FUNCTION_BLOCK HS_model
  (* Version 1.0, 2005-09-21, Goran Cengic, Chalmers *)
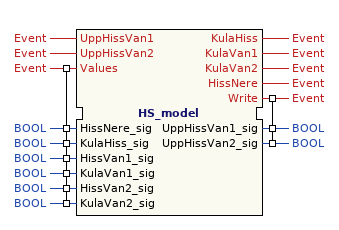
  EVENT_INPUT
    UppHissVan1;
    UppHissVan2;
    Values WITH KulaHiss_sig, HissVan1_sig, KulaVan1_sig, HissVan2_sig, KulaVan2_sig, HissNere_sig;
  END_EVENT
  EVENT_OUTPUT
    KulaHiss;
    KulaVan1;
    KulaVan2;
    HissNere;
    Write WITH UppHissVan1_sig, UppHissVan2_sig;
  END_EVENT
  VAR_INPUT
    HissNere_sig : BOOL;
    KulaHiss_sig : BOOL;
    HissVan1_sig : BOOL;
    KulaVan1_sig : BOOL;
    HissVan2_sig : BOOL;
    KulaVan2_sig : BOOL;
  END_VAR
  VAR_OUTPUT
    UppHissVan1_sig : BOOL;
    UppHissVan2_sig : BOOL;
  END_VAR
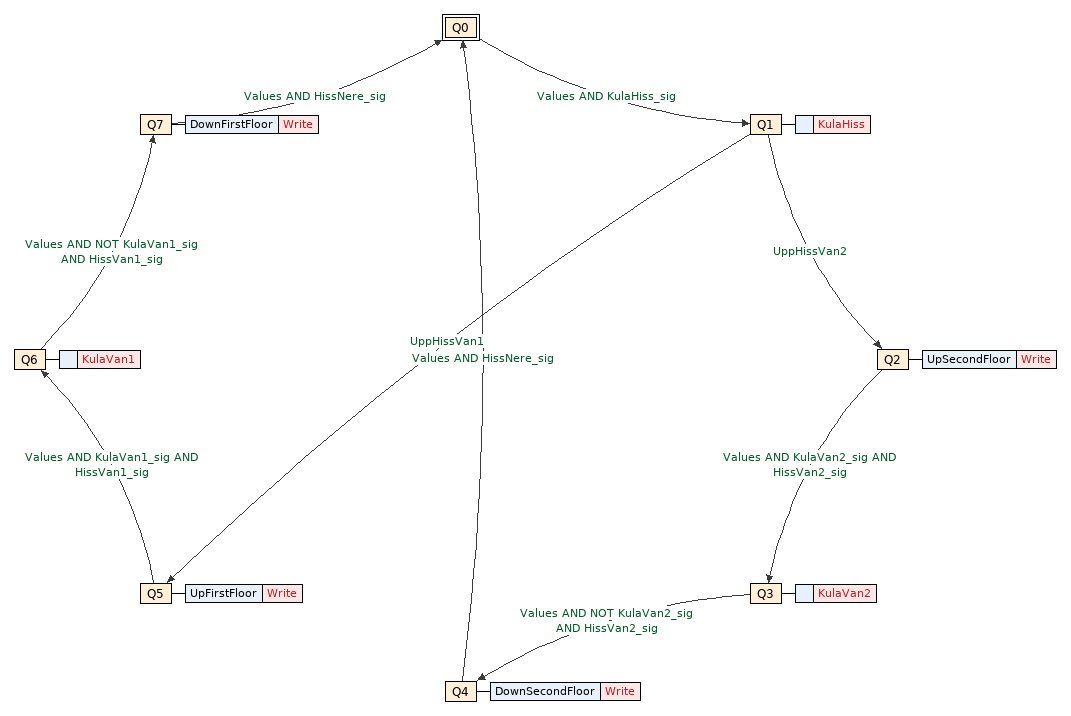
  EC_STATES
    Q0;
    Q1 : -> KulaHiss;
    Q2 : UpSecondFloor -> Write;
    Q3 : -> KulaVan2;
    Q4 : DownSecondFloor -> Write;
    Q5 : UpFirstFloor -> Write;
    Q6 : -> KulaVan1;
    Q7 : DownFirstFloor -> Write;
  END_STATES
  EC_TRANSITIONS
    Q0 TO Q1 := Values AND KulaHiss_sig;
    Q1 TO Q2 := UppHissVan2;
    Q1 TO Q5 := UppHissVan1;
    Q2 TO Q3 := Values AND KulaVan2_sig AND HissVan2_sig;
    Q3 TO Q4 := Values AND NOT KulaVan2_sig AND HissVan2_sig;
    Q4 TO Q0 := Values AND HissNere_sig;
    Q5 TO Q6 := Values AND KulaVan1_sig AND HissVan1_sig;
    Q6 TO Q7 := Values AND NOT KulaVan1_sig AND HissVan1_sig;
    Q7 TO Q0 := Values AND HissNere_sig;
  END_TRANSITIONS
  ALGORITHM UpSecondFloor IN Java:
		System.out.println("Elevator going up to second floor.");
		UppHissVan2_sig = true;
  END_ALGORITHM
  ALGORITHM DownSecondFloor IN Java:
		System.out.println("Elevator going down from second floor.");
		UppHissVan2_sig = false;
  END_ALGORITHM
  ALGORITHM UpFirstFloor IN Java:
		System.out.println("Elevator going up to first floor.");
		UppHissVan1_sig = true;
  END_ALGORITHM
  ALGORITHM DownFirstFloor IN Java:
		System.out.println("Elevator going down from first floor.");
		UppHissVan1_sig = false;
  END_ALGORITHM
END_FUNCTION_BLOCK
